(* Schneider Machine Expert - Basic project Hot Water Tank, file version 2.0.0.0 *)
(* ProjectInformations: Name=New project *)

HARDWARE
  Cpu 0: TM221CE16R
  EthernetConfiguration: NetworkName=M221, IpAllocationMode=FixedAddress, IpAddress=0.0.0.0, SubnetMask=0.0.0.0
  SerialLineConfiguration: Baud=Baud19200, Parity=ParityEven, DataBits=DataBits8, StopBits=StopBits1, PhysicalMedium=PhysicalMediumRs485, TransmissionMode=TransmissionModeModbusRtu, SlaveId=1, Addressing=SlaveAddressing
  MastTask: UsePeriodScanMode=false, PeriodScan=100
  FastTask: Period=255
  CpuBehavior: StartingMode=StartAsPreviousState, AutoSaveRamOnEeprom=true, WatchdogPeriod=250

SYMBOLS  (address, symbol, comment, settings)
  %I0.0       "Min. water level"
  %I0.2       "Lower water level"
  %I0.3       "Max. water level"
  %I0.4       "Min. Temperature"
  %I0.5       "Max. Temperature"
  %Q0.0       "Inlet valve"
  %Q0.1       "Inlet valve (slow)"
  %Q0.2       "Outlet valve"
  %Q0.3       "Heating"

POU New POU
  (* SectionNumber=1 *)

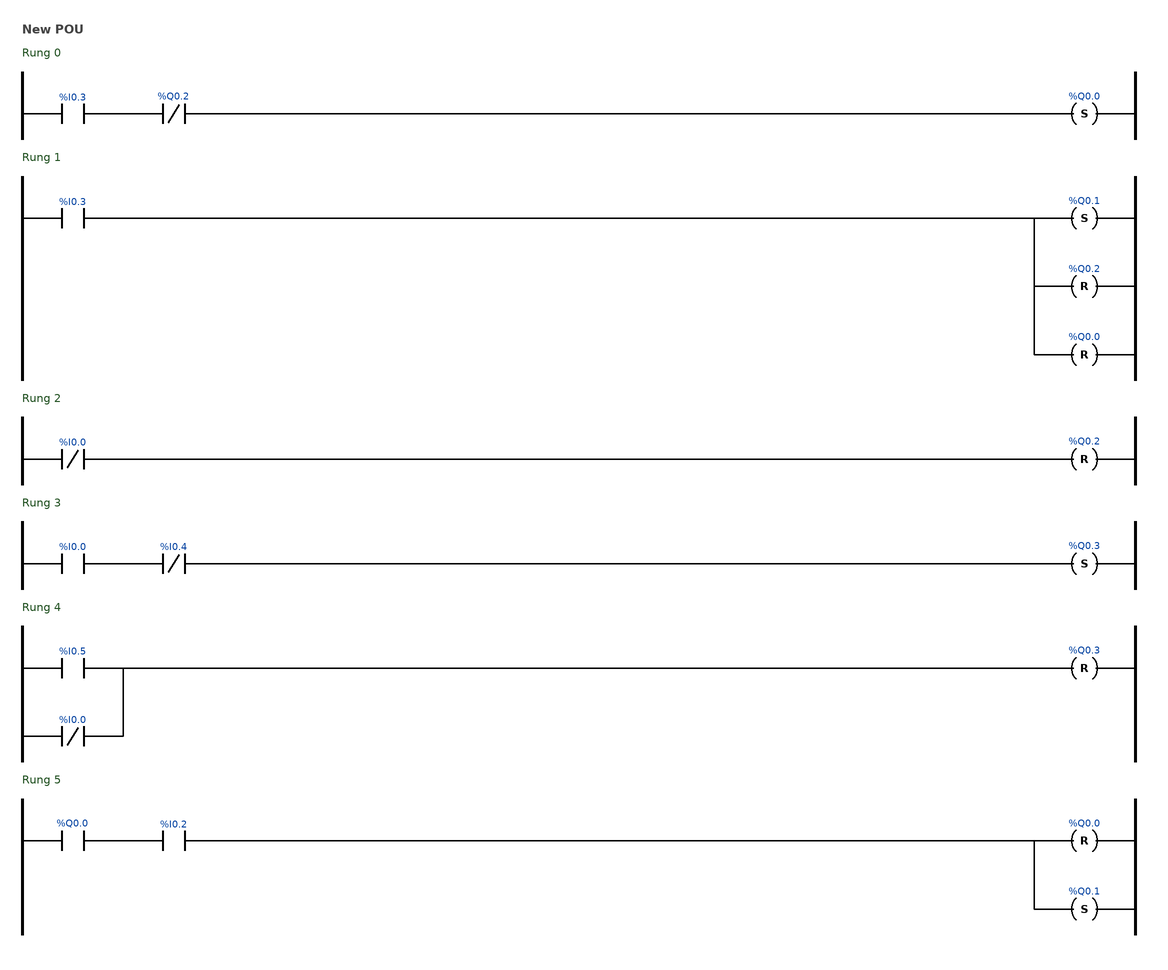

// Rung 0
  LD %I0.3
  ANDN %Q0.2
  S %Q0.0
  // as ST:
  //   IF %I0.3 AND NOT %Q0.2 THEN %Q0.0 := TRUE; END_IF;

// Rung 1
  LD %I0.3
  S %Q0.1
  R %Q0.2
  R %Q0.0
  // as ST:
  //   IF %I0.3 THEN %Q0.1 := TRUE; END_IF;
  //   IF %I0.3 THEN %Q0.2 := FALSE; END_IF;
  //   IF %I0.3 THEN %Q0.0 := FALSE; END_IF;

// Rung 2
  LDN %I0.0
  R %Q0.2
  // as ST:
  //   IF NOT %I0.0 THEN %Q0.2 := FALSE; END_IF;

// Rung 3
  LD %I0.0
  ANDN %I0.4
  S %Q0.3
  // as ST:
  //   IF %I0.0 AND NOT %I0.4 THEN %Q0.3 := TRUE; END_IF;

// Rung 4
  LD %I0.5
  ORN %I0.0
  R %Q0.3
  // as ST:
  //   IF %I0.5 OR NOT %I0.0 THEN %Q0.3 := FALSE; END_IF;

// Rung 5
  LD %Q0.0
  AND %I0.2
  R %Q0.0
  S %Q0.1
  // as ST:
  //   _t1 := %Q0.0 AND %I0.2;
  //   IF _t1 THEN %Q0.0 := FALSE; END_IF;
  //   IF _t1 THEN %Q0.1 := TRUE; END_IF;
